{attribute addProperty BoxType "EL1114-0000-0016"}
{attribute addProperty Id "ChannelAT %I*ARRAY[0..3] OF Channel_E4AEF59E3240WcStateAT %I*WcState_98A4DF7520.250InfoDataAT %I*InfoData_192954DE1620"}
{attribute addProperty CRC "2526129904"}
{attribute addProperty SizeInBites "50"}
{attribute addProperty SizeInBytes "6.25"}
TYPE EL1114_C1DCB3BD :
STRUCT
	{attribute addProperty Name "Channel"}
	Channel : ARRAY[0..3] OF Channel_E4AEF59E;
	{attribute addProperty Name "WcState"}
	WcState : WcState_98A4DF75;
	{attribute addProperty Name "InfoData"}
	InfoData : InfoData_192954DE;
END_STRUCT
END_TYPE

(* stored: Version 1.2.0.0, ProductVersion 3.1.4024.9
   DUT EL1114_C1DCB3BD: Id {6eb50d25-c875-4074-abdb-2fb32c855c5f} *)
